{attribute 'GeneratedUsingTerminal: EL3061-0000-0016'}
{attribute addProperty BoxType "EL3061-0000-0016"}
{attribute addProperty Id "AI_StandardAT %I*AI_Standard_EA9DF21E9WcStateAT %I*WcState_9091E0EB2InfoDataAT %I*InfoData_94A18F5E2"}
{attribute addProperty CRC "2525071622"}
{attribute addProperty Size "13"}
TYPE EL3061_96818906 EXTENDS EtcSlaveTerminalBase_947E5A46 :
STRUCT
	{attribute addProperty Name "AI_Standard"}
	AI_Standard : AI_Standard_EA9DF21E;
	{attribute addProperty Name "WcState"}
	WcState : WcState_9091E0EB;
	{attribute addProperty Name "InfoData"}
	InfoData : InfoData_94A18F5E;
END_STRUCT
END_TYPE

(* stored: Version 1.2.0.0, ProductVersion 3.1.4024.9
   DUT EL3061_96818906: Id {8beb7e9c-ad59-472e-8928-51ba8053fa27} *)
